FUNCTION F_GetSysTime : ULINT
VAR_INPUT
END_VAR
VAR
	GetSystemTime:GETSYSTEMTIME;
END_VAR

GetSystemTime(timeLoDW=>,timeHiDW=>);
F_GetSysTime:=UDINT_TO_ULINT(GetSystemTime.timeHiDW)*4294967296+UDINT_TO_ULINT(GetSystemTime.timeLoDW)/10000;

END_FUNCTION

(* stored: Version 1.1.0.1, ProductVersion 3.1.4024.6
   POU F_GetSysTime: Id {db418080-88cc-4e5d-bad1-a178be8bfab5}, SpecialFunc None *)
